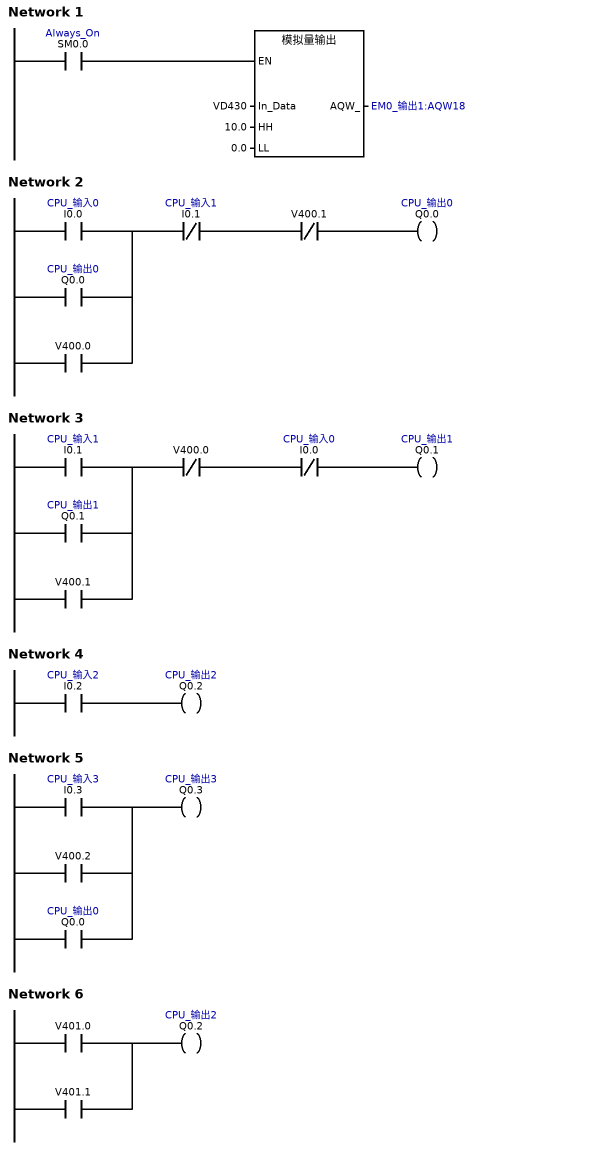
[picture p24: SBR13 networks 1-6]
Network 1
LD     Always_On:SM0.0
CALL   模拟量输出:SBR3, VD430, 10.0, 0.0, EM0_输出1:AQW18
Network 2
LD     CPU_输入0:I0.0
O      CPU_输出0:Q0.0
O      V400.0
AN     CPU_输入1:I0.1
AN     V400.1
=      CPU_输出0:Q0.0
Network 3
LD     CPU_输入1:I0.1
O      CPU_输出1:Q0.1
O      V400.1
AN     V400.0
AN     CPU_输入0:I0.0
=      CPU_输出1:Q0.1
Network 4
LD     CPU_输入2:I0.2
=      CPU_输出2:Q0.2
Network 5
LD     CPU_输入3:I0.3
O      V400.2
O      CPU_输出0:Q0.0
=      CPU_输出3:Q0.3
Network 6
LD     V401.0
O      V401.1
=      CPU_输出2:Q0.2
END_SUBROUTINE_BLOCK

SUBROUTINE_BLOCK 循环:SBR14
TITLE=
BEGIN
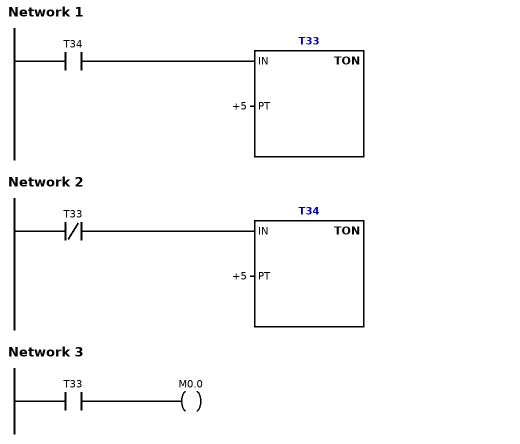
Network 1
LD     T34
TON    T33, +5
Network 2
LDN    T33
TON    T34, +5
Network 3
LD     T33
=      M0.0
END_SUBROUTINE_BLOCK

INTERRUPT_BLOCK INT_0:INT0
TITLE=中断例程注释
BEGIN
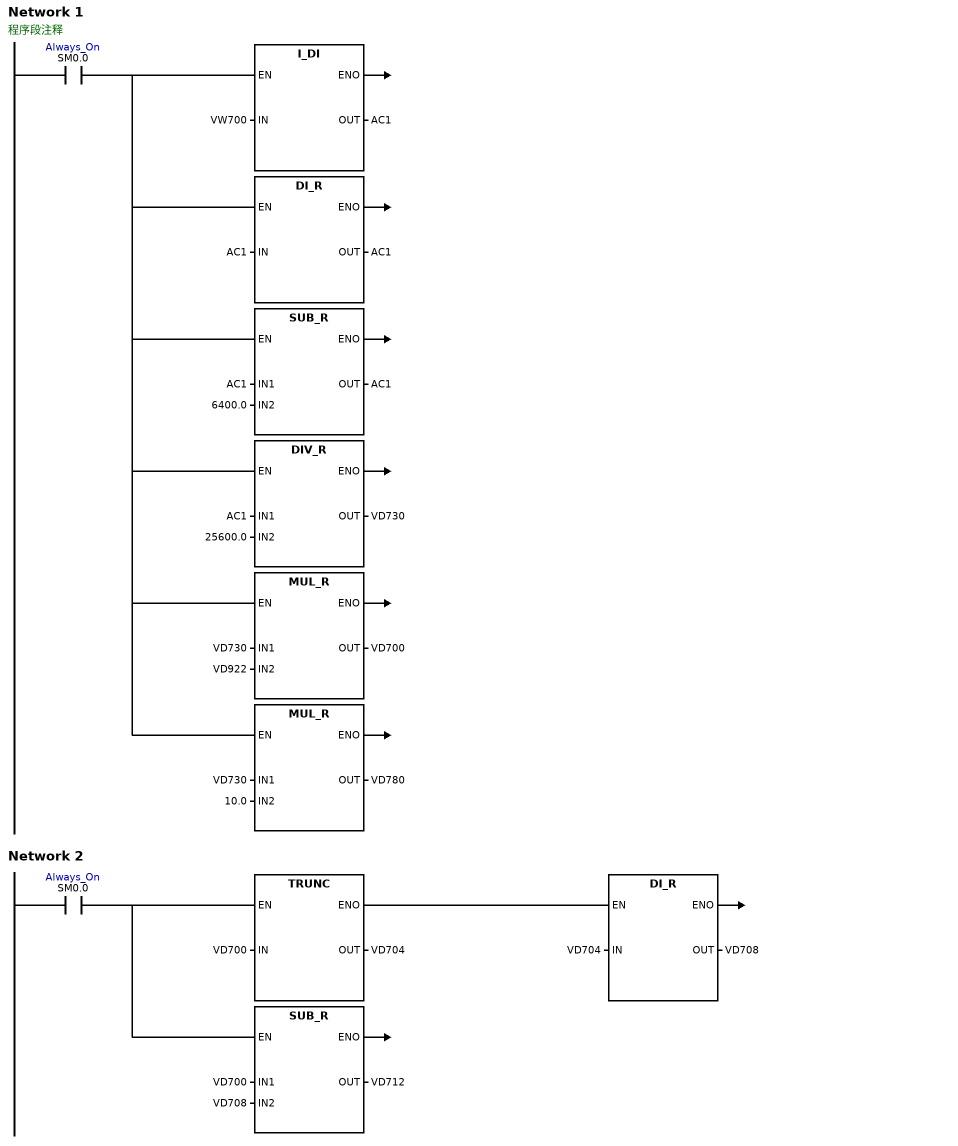
Network 1
// 程序段注释
LD     Always_On:SM0.0
ITD    VW700, AC1
DTR    AC1, AC1
-R     6400.0, AC1
MOVR   AC1, VD730
/R     25600.0, VD730
MOVR   VD730, VD700
*R     VD922, VD700
MOVR   VD730, VD780
*R     10.0, VD780
Network 2
LD     Always_On:SM0.0
LPS
TRUNC  VD700, VD704
AENO
DTR    VD704, VD708
LPP
MOVR   VD700, VD712
-R     VD708, VD712
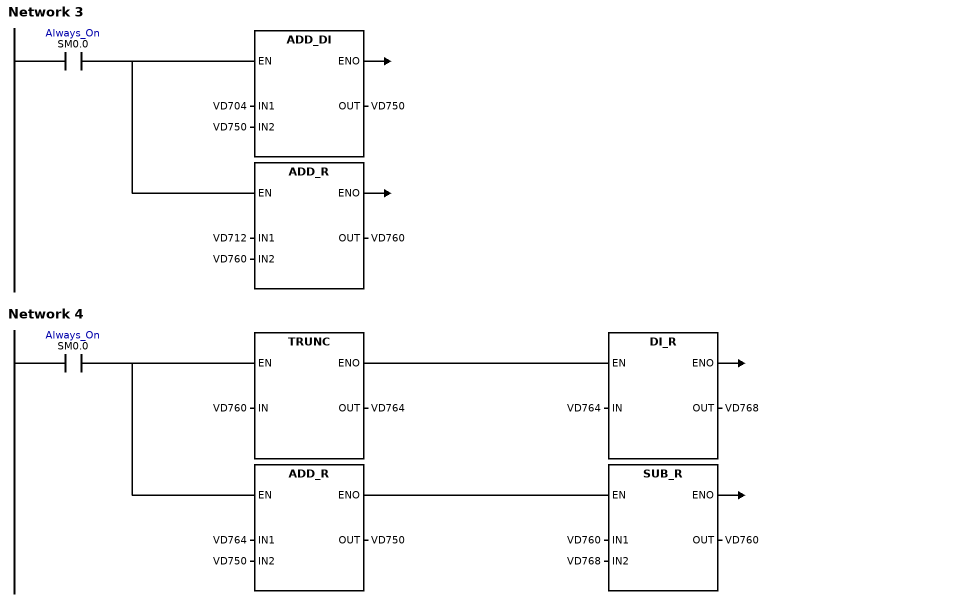
Network 3
LD     Always_On:SM0.0
+D     VD704, VD750
+R     VD712, VD760
Network 4
LD     Always_On:SM0.0
LPS
TRUNC  VD760, VD764
AENO
DTR    VD764, VD768
LPP
+R     VD764, VD750
AENO
-R     VD768, VD760
END_INTERRUPT_BLOCK
